FUNCTION_BLOCK CiA_DS402Controlword
VAR_INPUT
	SwitchOn 				: BOOL;	// BIT 0 
	EnableVoltage 			: BOOL := TRUE; // Bit 1  
	QuickStopOK 			: BOOL := TRUE; // Bit 2 inverse signal / TRUE = RUN -
	EnableOperation 		: BOOL; // Bit 3 
//	Operation mode specific Bit 4 	: BOOL; // Bit 4
//	Operation mode specific Bit 5 	: BOOL; // Bit 5
//	Operation mode specific Bit 6 	: BOOL; // Bit 6
	FaultReset 				: BOOL; // Bit 7 
	Halt 					: BOOL; // Bit 8 - Pauses the drive in all modes
//	Operation mode specific Bit 9 	: BOOL; // Bit 9 - 
//	Reserved Bit 10 	: BOOL; // Bit 10
//	Manufacturere specific Bit 11 	: BOOL; // Bit 11
//	Manufacturere specific Bit 12 	: BOOL; // Bit 12
//	Manufacturere specific Bit 13 	: BOOL; // Bit 13
//	Manufacturere specific Bit 14 	: BOOL; // Bit 14
//	Manufacturere specific Bit 15 	: BOOL; // Bit 15	
END_VAR
VAR_OUTPUT
	Cmd						:	eCiA_DS402_CONTROL_CMD;
END_VAR
VAR
END_VAR

;

METHOD PUBLIC createControlword : BOOL
VAR_INPUT
	StatusState												: 	eCiA_DS402_STATUS_STATE;
END_VAR
VAR_IN_OUT
	Controlword												:	UINT;
END_VAR
(* work local state machine for control ****************************************************)
	CASE StatusState OF
	eCiA_DS402_STATUS_STATE.NOT_READY_TO_SWITCH_ON:
		Controlword.0										:= FALSE;
		Controlword.1										:= FALSE;
		Controlword.2										:= FALSE;
		Controlword.3										:= FALSE;
		Cmd													:= eCiA_DS402_CONTROL_CMD.DISABLE_VOLTAGE;
		
	eCiA_DS402_STATUS_STATE.SWITCH_ON_DISABLED:
		IF EnableVoltage
		THEN //back to "not ready to switch on"
			Controlword.0									:= FALSE;
			Controlword.1									:= TRUE;
			Controlword.2									:= TRUE;
			Controlword.3									:= FALSE;
			Cmd												:= eCiA_DS402_CONTROL_CMD.SHUTDOWN;
		ELSE //To "Ready to switch on"
			Controlword.0									:= FALSE;
			Controlword.1									:= FALSE;
			Controlword.2									:= FALSE;
			Controlword.3									:= FALSE;
			Cmd												:= eCiA_DS402_CONTROL_CMD.DISABLE_VOLTAGE;
		END_IF
		
	eCiA_DS402_STATUS_STATE.READY_TO_SWITCH_ON:
		IF NOT EnableVoltage
		THEN //Back to switched on disabled
			Controlword.0									:= FALSE;
			Controlword.1									:= FALSE;
			Controlword.2									:= FALSE;
			Controlword.3									:= FALSE;
			Cmd												:= eCiA_DS402_CONTROL_CMD.DISABLE_VOLTAGE;
		ELSIF SwitchOn
		THEN //To switched on
			Controlword.0									:= TRUE;
			Controlword.1									:= TRUE;
			Controlword.2									:= QuickStopOK;
			Controlword.3									:= FALSE;
			Cmd												:= eCiA_DS402_CONTROL_CMD.SWITCH_ON;	
		ELSE
			Controlword.0									:= FALSE;
			Controlword.1									:= TRUE;
			Controlword.2									:= QuickStopOK;
			Controlword.3									:= FALSE;
			Cmd												:= eCiA_DS402_CONTROL_CMD.SHUTDOWN;			
		END_IF	
		
	eCiA_DS402_STATUS_STATE.SWITCHED_ON:
		IF NOT EnableVoltage
		THEN //Back to switched on disabled
			Controlword.0									:= FALSE;
			Controlword.1									:= FALSE;
			Controlword.2									:= FALSE;
			Controlword.3									:= FALSE;
			Cmd												:= eCiA_DS402_CONTROL_CMD.DISABLE_VOLTAGE;
		ELSIF NOT SwitchOn
		THEN
			Controlword.0									:= FALSE;
			Controlword.1									:= TRUE;
			Controlword.2									:= QuickStopOK;
			Controlword.3									:= FALSE;
			Cmd												:= eCiA_DS402_CONTROL_CMD.SHUTDOWN;

		ELSIF EnableOperation
		THEN // To operation enabled
			Controlword.0									:= TRUE;
			Controlword.1									:= TRUE;
			Controlword.2									:= QuickStopOK;
			Controlword.3									:= TRUE;
			Cmd												:= SEL(QuickStopOK,eCiA_DS402_CONTROL_CMD.QUICK_STOP,eCiA_DS402_CONTROL_CMD.ENABLE_OPERATION);												
		ELSE
			Controlword.0									:= TRUE;
			Controlword.1									:= TRUE;
			Controlword.2									:= QuickStopOK;
			Controlword.3									:= FALSE;
			Cmd												:= eCiA_DS402_CONTROL_CMD.SWITCH_ON;						
		END_IF
		
	eCiA_DS402_STATUS_STATE.OPERATION_ENABLED:
		IF NOT EnableVoltage
		THEN //Back to switch on disabled
			Controlword.0									:= FALSE;
			Controlword.1									:= FALSE;
			Controlword.2									:= FALSE;
			Controlword.3									:= FALSE;
			Cmd												:= eCiA_DS402_CONTROL_CMD.DISABLE_VOLTAGE;
		ELSIF NOT SwitchOn		
		THEN // back to ready to switch on 
			Controlword.0									:= FALSE;
			Controlword.1									:= TRUE;
			Controlword.2									:= QuickStopOK;
			Controlword.3									:= FALSE;
			Cmd												:= eCiA_DS402_CONTROL_CMD.SHUTDOWN;	
		ELSIF NOT EnableOperation 
		THEN //go back to switched on
			Controlword.0									:= TRUE;
			Controlword.1									:= TRUE;
			Controlword.2									:= QuickStopOK;
			Controlword.3									:= FALSE;
			Cmd												:= eCiA_DS402_CONTROL_CMD.SWITCH_ON;
		ELSE
			Controlword.0									:= TRUE;
			Controlword.1									:= TRUE;
			Controlword.2									:= QuickStopOK;
			Controlword.3									:= TRUE;
			Cmd												:= SEL(QuickStopOK,eCiA_DS402_CONTROL_CMD.QUICK_STOP,eCiA_DS402_CONTROL_CMD.ENABLE_OPERATION);												
		END_IF
		
	eCiA_DS402_STATUS_STATE.QUICK_STOP_ACTIVE:
		IF NOT EnableVoltage
		THEN //Back to switch on disabled
			Controlword.0									:= FALSE;
			Controlword.1									:= FALSE;
			Controlword.2									:= FALSE;
			Controlword.3									:= FALSE;
			Cmd												:= eCiA_DS402_CONTROL_CMD.DISABLE_VOLTAGE;
		ELSIF NOT SwitchOn		
		THEN // back to ready to switch on 
			Controlword.0									:= FALSE;
			Controlword.1									:= TRUE;
			Controlword.2									:= QuickStopOK;
			Controlword.3									:= FALSE;
			Cmd												:= eCiA_DS402_CONTROL_CMD.SHUTDOWN;		
		ELSIF NOT EnableOperation 
		THEN //go back to switched on
			Controlword.0									:= TRUE;
			Controlword.1									:= TRUE;
			Controlword.2									:= QuickStopOK;
			Controlword.3									:= FALSE;
			Cmd												:= eCiA_DS402_CONTROL_CMD.SWITCH_ON;
		ELSE
			Controlword.0									:= TRUE;
			Controlword.1									:= TRUE;
			Controlword.2									:= QuickStopOK;
			Controlword.3									:= TRUE;
			Cmd												:= SEL(QuickStopOK,eCiA_DS402_CONTROL_CMD.QUICK_STOP,eCiA_DS402_CONTROL_CMD.ENABLE_OPERATION);												
		END_IF
		
	eCiA_DS402_STATUS_STATE.FAULT_ACTIVE:
		IF NOT EnableVoltage
		THEN //back to "not ready to switch on"
			Controlword.0									:= FALSE;
			Controlword.1									:= FALSE;
			Controlword.2									:= FALSE;
			Controlword.3									:= FALSE;
			Cmd												:= eCiA_DS402_CONTROL_CMD.DISABLE_VOLTAGE;
		ELSE //To "Ready to switch on"
			Controlword.0									:= FALSE;
			Controlword.1									:= TRUE;
			Controlword.2									:= QuickStopOK;
			Controlword.3									:= FALSE;
			Cmd												:= eCiA_DS402_CONTROL_CMD.SHUTDOWN;	
		END_IF
		
	eCiA_DS402_STATUS_STATE.FAULT_REACTION_ACTIVE:
		;	
	END_CASE
	
(* Write controlword ********************************************************)
	Controlword.7											:= FaultReset; 
	createControlword										:= TRUE;
(*****************************************************************************)
END_METHOD

END_FUNCTION_BLOCK

(* stored: Version 1.1.0.1, ProductVersion 3.1.4024.12
   POU CiA_DS402Controlword: Id {a10ef42a-c64d-4e19-9c16-13d4d0845468}, SpecialFunc None
   Method createControlword: Id {af09360e-7f59-4703-9767-f0a295d44be2} *)
